{attribute 'GeneratedUsingTerminal: EK1100-0000-0018'}
{attribute addProperty BoxType "EK1100-0000-0018"}
{attribute addProperty Id "Beckhoff_EPP9xxxEK1122Beckhoff_EPP9xxxEK1122_FD80CF4A86"}
{attribute addProperty CRC "733959567"}
{attribute addProperty Size "86"}
TYPE Beckhoff_EPP9xxx_2BBF558F EXTENDS EK1100_1FC0878B :
STRUCT
	{attribute addProperty Name "Beckhoff_EPP9xxxEK1122"}
	{attribute addProperty PreviousPort "Beckhoff EPP9xxx : B"}
	Beckhoff_EPP9xxxEK1122 : Beckhoff_EPP9xxxEK1122_FD80CF4A;
END_STRUCT
END_TYPE

(* stored: Version 1.2.0.0, ProductVersion 3.1.4024.9
   DUT Beckhoff_EPP9xxx_2BBF558F: Id {03226ed7-e1ee-4aac-a2aa-a625f396946f} *)
